{attribute 'qualified_only'}
{attribute 'strict'}
{attribute 'to_string'}
TYPE TASK_RUNNING_STATE :
(
	BUSY := 0,
	DONE := 1,
	ABORTED := 2
);
END_TYPE

(* stored: Version 1.1.0.1
   DUT TASK_RUNNING_STATE: Id {608d5f96-937e-4934-ad17-0359734bd53a} *)
